Fanuc KAREL source: kt00212.KL

-- PROVISIONAL review KL for V1013-1; original PC SHA256 3a5f1d0209df6a61c84456d4789f788d33a7ee22e30bd293cbfa9afa0a018962
-- Incomplete behavior may be omitted. Consult companion uncertainty JSON. Do not deploy.
PROGRAM KT00212
%NOLOCKGROUP
VAR
  I2 : INTEGER
  OUT : INTEGER
-- UNRESOLVED_DECL Y1 type=002018
BEGIN
  -- UNRESOLVED_PC offsets 5-19; opcodes 2E,22,9D,33,B2
  -- UNRESOLVED_PC offsets 24-35; opcodes 2E,23
  -- UNRESOLVED_PC offsets 40-62; opcodes 22,9D,33,B1,21,46,23
  -- UNRESOLVED_PC offsets 67-71; opcodes 7F
END KT00212
